Fanuc KAREL source: NC0033.KL

-- PROVISIONAL review KL for V770-1; original PC SHA256 a3ecf154efebf418fca100c1194ed35ffaf9051164ed4d70326c21c5cfb19fdb
-- Incomplete behavior may be omitted. Consult companion uncertainty JSON. Do not deploy.
PROGRAM NC0033
%NOLOCKGROUP
-- UNRESOLVED_LOCAL_POOL 1 cells at code offset 3; source declarations unknown
-- DIRECT_LOCAL_WORD_ACCESS alone does not prove INTEGER, REAL, or BOOLEAN
BEGIN
  -- UNRESOLVED_PC offsets 0-8; opcodes 2B,2C,7B
  -- UNRESOLVED_PC offsets 13-20; opcodes 9D,23
  -- UNRESOLVED_PC offsets 25-42; opcodes 21,40,41,42
  -- UNRESOLVED_PC offsets 47-81; opcodes 21,2E,52,23,7A,40,41,42
  -- UNRESOLVED_PC offsets 86-110; opcodes 21,2E,52,23,7A,43
  -- UNRESOLVED_PC offsets 115-132; opcodes 21,40,41,42
  -- UNRESOLVED_PC offsets 137-171; opcodes 21,2E,52,23,7A,40,41,42
  -- UNRESOLVED_PC offsets 176-200; opcodes 21,2E,52,23,7A,43
  -- UNRESOLVED_PC offsets 205-219; opcodes 21,9D,52,23
  -- UNRESOLVED_PC offsets 234-238; opcodes 7F
  -- UNRESOLVED_PC offsets 243-247; opcodes 27,AA
  -- UNRESOLVED_PC offsets 252-256; opcodes 7F
END NC0033
